    // reduced muon Compton wavelength (m)
    // Uncertainty: 4.2e-23
    fReducedMuonComptonWavelength_in_m : LREAL := 1.867594306e-15;
    fReducedMuonComptonWavelength_in_m_Units : STRING := 'm';
    fReducedMuonComptonWavelength_in_m_Uncertainty : LREAL := 4.2e-23;
    
    // reduced neutron Compton wavelength (m)
    // Uncertainty: 1.2e-25
    fReducedNeutronComptonWavelength_in_m : LREAL := 2.1001941552e-16;
    fReducedNeutronComptonWavelength_in_m_Units : STRING := 'm';
    fReducedNeutronComptonWavelength_in_m_Uncertainty : LREAL := 1.2e-25;
    
    // reduced Planck constant (J s)
    fReducedPlanckConstant_in_J_s : LREAL := 1.054571817e-34;
    fReducedPlanckConstant_in_J_s_Units : STRING := 'J s';
    
    // reduced Planck constant in eV s (eV s)
    fReducedPlanckConstantInEVS_in_eV_s : LREAL := 6.582119569e-16;
    fReducedPlanckConstantInEVS_in_eV_s_Units : STRING := 'eV s';
    
    // reduced Planck constant times c in MeV fm (MeV fm)
    fReducedPlanckConstantTimesCInMeVFm_in_MeV_fm : LREAL := 197.3269804;
    fReducedPlanckConstantTimesCInMeVFm_in_MeV_fm_Units : STRING := 'MeV fm';
    
    // reduced proton Compton wavelength (m)
    // Uncertainty: 6.4e-26
    fReducedProtonComptonWavelength_in_m : LREAL := 2.10308910336e-16;
    fReducedProtonComptonWavelength_in_m_Units : STRING := 'm';
    fReducedProtonComptonWavelength_in_m_Uncertainty : LREAL := 6.4e-26;
    
    // reduced tau Compton wavelength (m)
    // Uncertainty: 7.5e-21
    fReducedTauComptonWavelength_in_m : LREAL := 1.110538e-16;
    fReducedTauComptonWavelength_in_m_Units : STRING := 'm';
    fReducedTauComptonWavelength_in_m_Uncertainty : LREAL := 7.5e-21;
    
    // shielded helion gyromag. ratio in MHz/T (MHz T^-1)
    // Uncertainty: 3.8e-07
    fShieldedHelionGyromag_RatioInMHz_T_in_MHz_T_1 : LREAL := 32.43409942;
    fShieldedHelionGyromag_RatioInMHz_T_in_MHz_T_1_Units : STRING := 'MHz T^-1';
    fShieldedHelionGyromag_RatioInMHz_T_in_MHz_T_1_Uncertainty : LREAL := 3.8e-07;
    
    // shielded proton gyromag. ratio in MHz/T (MHz T^-1)
    // Uncertainty: 4.6e-07
    fShieldedProtonGyromag_RatioInMHz_T_in_MHz_T_1 : LREAL := 42.57638474;
    fShieldedProtonGyromag_RatioInMHz_T_in_MHz_T_1_Units : STRING := 'MHz T^-1';
    fShieldedProtonGyromag_RatioInMHz_T_in_MHz_T_1_Uncertainty : LREAL := 4.6e-07;
    
    // shielding difference of d and p in HD
    // Uncertainty: 2e-11
    fShieldingDifferenceOfDAndPInHD : LREAL := 2.02e-08;
    fShieldingDifferenceOfDAndPInHD_Uncertainty : LREAL := 2e-11;
    
    // shielding difference of t and p in HT
    // Uncertainty: 2e-11
    fShieldingDifferenceOfTAndPInHT : LREAL := 2.414e-08;
    fShieldingDifferenceOfTAndPInHT_Uncertainty : LREAL := 2e-11;
    
    // tau energy equivalent (MeV)
    // Uncertainty: 0.12
    fTauEnergyEquivalent_in_MeV : LREAL := 1776.86;
    fTauEnergyEquivalent_in_MeV_Units : STRING := 'MeV';
    fTauEnergyEquivalent_in_MeV_Uncertainty : LREAL := 0.12;
    
    // triton relative atomic mass
    // Uncertainty: 1.2e-10
    fTritonRelativeAtomicMass : LREAL := 3.01550071621;
    fTritonRelativeAtomicMass_Uncertainty : LREAL := 1.2e-10;
    
    // triton to proton mag. mom. ratio
    // Uncertainty: 2.1e-09
    fTritonToProtonMag_Mom_Ratio : LREAL := 1.0666399191;
    fTritonToProtonMag_Mom_Ratio_Uncertainty : LREAL := 2.1e-09;
    
    // vacuum electric permittivity (F m^-1)
    // Uncertainty: 1.3e-21
    fVacuumElectricPermittivity_in_F_m_1 : LREAL := 8.8541878128e-12;
    fVacuumElectricPermittivity_in_F_m_1_Units : STRING := 'F m^-1';
    fVacuumElectricPermittivity_in_F_m_1_Uncertainty : LREAL := 1.3e-21;
    
    // vacuum mag. permeability (N A^-2)
    // Uncertainty: 1.9e-16
    fVacuumMag_Permeability_in_N_A_2 : LREAL := 1.25663706212e-06;
    fVacuumMag_Permeability_in_N_A_2_Units : STRING := 'N A^-2';
    fVacuumMag_Permeability_in_N_A_2_Uncertainty : LREAL := 1.9e-16;
    
    // W to Z mass ratio
    // Uncertainty: 0.00017
    fWToZMassRatio : LREAL := 0.88153;
    fWToZMassRatio_Uncertainty : LREAL := 0.00017;
    
END_VAR

(* stored: Version 1.1.0.1, ProductVersion 3.1.4024.4
   GVL GVL_PhysicalConstants: Id {bf9314b5-5147-8274-e829-1de2bc69af7d}, SpecialFunc None *)
